FUNCTION_BLOCK Tiefpassfilter
VAR_INPUT
	x : REAL;
	h : REAL;
	tau : REAL;
END_VAR
VAR_OUTPUT
	y : REAL;
END_VAR
VAR
	xm : REAL;
	ym : REAL;
END_VAR

y := (h/tau)*xm-((h/tau)-1)*ym;
ym := y;
xm := x;

END_FUNCTION_BLOCK

(* stored: Version 1.1.0.1, ProductVersion 3.1.4024.13
   POU Tiefpassfilter: Id {eeeb2314-48ff-4d6f-ab45-929f1a32f6b6}, SpecialFunc None *)
